{attribute 'GeneratedUsingTerminal: EL6201-0000-0017'}
{attribute addProperty BoxType "EL6201-0000-0017"}
{attribute addProperty Id "ASI_Inputs_DeviceAT %I*ASI_Inputs_Device_7F2828A5248ASI_StatusAT %I*ASI_Status_8C8FBBB411ASI_Outputs_DeviceAT %Q*ASI_Outputs_Device_16036E19248ASI_ControlAT %Q*ASI_Control_F45BBE2B5WcStateAT %I*WcState_9091E0EB2InfoDataAT %I*InfoData_32EB74EA10"}
{attribute addProperty CRC "318525277"}
{attribute addProperty Size "524"}
TYPE EL6201_12FC4F5D EXTENDS EtcSlaveTerminalBase_947E5A46 :
STRUCT
	{attribute addProperty Name "ASI_Inputs_Device"}
	ASI_Inputs_Device : ASI_Inputs_Device_7F2828A5;
	{attribute addProperty Name "ASI_Status"}
	ASI_Status : ASI_Status_8C8FBBB4;
	{attribute addProperty Name "ASI_Outputs_Device"}
	ASI_Outputs_Device : ASI_Outputs_Device_16036E19;
	{attribute addProperty Name "ASI_Control"}
	ASI_Control : ASI_Control_F45BBE2B;
	{attribute addProperty Name "WcState"}
	WcState : WcState_9091E0EB;
	{attribute addProperty Name "InfoData"}
	InfoData : InfoData_32EB74EA;
END_STRUCT
END_TYPE

(* stored: Version 1.2.0.0, ProductVersion 3.1.4024.9
   DUT EL6201_12FC4F5D: Id {2f203285-cb6e-4983-bfa9-a377c8e16063} *)
